// Mitsubishi GX Works2 project: 17   PLC: FX3G

// task Task_01 (event TRUE, interval 0, priority 31): POU_01

PROGRAM POU_01
VAR
  wstep : INT;
  wstep2 : INT;
  wstep3 : INT;
  ton1 : TON;
  ton2 : TON;
END_VAR
IF M8002 THEN
	wstep := 0;
	wstep2 := 0;
	wstep3 := 0;
END_IF;

CASE wstep OF 
	0:
		IF M5 THEN
			wstep := 20;
		END_IF;
		
	20:
		Y1 := FALSE;
		Y2 := TRUE;
		Y3 := TRUE;
		ton1(IN := NOT ton1.Q, PT := T#8s);
		IF ton1.Q THEN
			wstep := 21;
		END_IF;
	
	21:
		Y3 := M8013;
		ton1(IN := NOT ton1.Q, PT := T#3s);
		IF ton1.Q THEN
			wstep := 22;
		END_IF;
		
	22:
		Y3 := FALSE;
		Y4 := TRUE;
		ton1(IN := NOT ton1.Q, PT := T#3s);
		IF ton1.Q THEN
			wstep := 23;
		END_IF;
		
	23:
		Y0 := TRUE;
		Y4 := FALSE;
		Y5 := TRUE;
		ton1(IN := NOT ton1.Q, PT := T#8s);
		IF ton1.Q THEN
			wstep := 24;
		END_IF;
	
	24:
		Y0 := M8013;
		ton1(IN := NOT ton1.Q, PT := T#3s);
		IF ton1.Q THEN
			wstep := 22;
		END_IF;
		
	25:	
		Y0 := FALSE;
		Y1 := TRUE;
		ton1(IN := NOT ton1.Q, PT := T#3s);
		IF ton1.Q THEN
			wstep := 20;
		END_IF;
END_CASE;
END_PROGRAM
